# EPICS substitutions: evrSupport/Db/ioc/IOC-IN20-AM01evr.substitutions
#==============================================================================
#
# Abs:  LCLS EVR IOC records for IN20 AM01
#
# Name: IOC-IN20-AM01evr.substitutions
#
#==============================================================================
#
file evrMCXX.db
{
pattern { DEVICE        }
	{ EVR:IN20:AM01 }
}
